// TwinCAT 3 PLC project Untitled1
// ProgramVersion: 3.1.4023.0
// libraries:
//   Tc2_Standard, * (Beckhoff Automation GmbH)
//   Tc2_System, * (Beckhoff Automation GmbH)
//   Tc3_Module, * (Beckhoff Automation GmbH)
// project tree:
//   / PlcTask.TcTTO
//   POUs/ MAIN.TcPOU
//   SUBMODULES/submodule1/POUs/ MAIN_1.TcPOU (not stored)
//   SUBMODULES/submodule2/POUs/ MAIN_2.TcPOU
// real-time tasks:
//   TASK PlcTask: cycle T#10ms, priority 20, ADS port 350

CONFIGURATION Untitled1
    RESOURCE PLC ON TwinCAT3
        TASK PlcTask(INTERVAL := T#10ms, PRIORITY := 20);
        PROGRAM MAIN WITH PlcTask : MAIN;
    END_RESOURCE
END_CONFIGURATION

// ---- POUs/MAIN.TcPOU
PROGRAM MAIN
VAR
	counter:INT:=0;
END_VAR

counter:=counter+1;

MAIN_1();
MAIN_2();

END_PROGRAM

// ---- SUBMODULES/submodule2/POUs/MAIN_2.TcPOU
PROGRAM MAIN_2
VAR
	counter_2:INT:=0;
END_VAR

counter_2:=counter_2+1;

END_PROGRAM
